(* CODESYS project gpio_lib.library
   Author: prg
   Version: 3.5.10.40
   Description: the operation of cyber gpio
   Title: cyber gpio
   Company: cyber

Project tree, tasks and I/O mapping:
  function set_gpio_value [ST]
*)

// set_gpio_value
FUNCTION set_gpio_value : INT
VAR_INPUT
	num :INT;
	value :INT;
END_VAR
VAR
END_VAR

END_FUNCTION
